{attribute addProperty BoxType "EL5072-0000-0016"}
{attribute addProperty Id "StatusAT %I*Status_E10353591621PositionAT %I*DINT3241Latch_valueAT %I*DINT3242"}
{attribute addProperty CRC "4044371903"}
{attribute addProperty SizeInBites "80"}
{attribute addProperty SizeInBytes "10"}
TYPE IND_Inputs_Channel_F11037BF :
STRUCT
	{attribute addProperty Name "Status"}
	Status AT %I* : Status_E1035359;
	{attribute addProperty Name "Position"}
	Position AT %I* : DINT;
	{attribute addProperty Name "Latch_value"}
	Latch_value AT %I* : DINT;
END_STRUCT
END_TYPE

(* stored: Version 1.2.0.0, ProductVersion 3.1.4024.9
   DUT IND_Inputs_Channel_F11037BF: Id {47d111d9-2c5f-4a19-835f-5e5b5e15e0a2} *)
